Fanuc KAREL source: GET_REG.kl

PROGRAM T
%NOLOCKGROUP
VAR
 v0 : INTEGER
 v1 : BOOLEAN
 v2 : INTEGER
 v3 : REAL
 v4 : INTEGER
BEGIN
 GET_REG(v0, v1, v2, v3, v4)
END T
